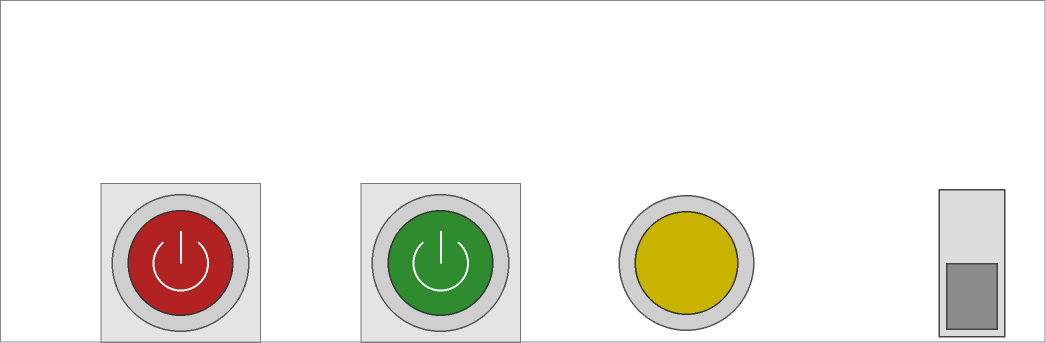
VISUALIZATION Visualization  // 1046x343
    PowerSwitch (83,183 195x160), variable: MAIN.bStopButton, behaviour: TOGGLE, style: Switch-PowerSwitch-Red
    PowerSwitch (343,183 195x160), variable: MAIN.bStartButton, behaviour: TOGGLE, style: Switch-PowerSwitch-Green
    Lamp1 (608,183 157x160), variable: MAIN.bMotor, style: Lamp-Lamp1-Yellow
    DipSwitch (898,183 148x160), variable: MAIN.bLimitSwitch, behaviour: TOGGLE, style: Switch-DipSwitch-Gray
END_VISUALIZATION

(* stored: Version 1.1.0.1
   Visu Visualization: Id {09181a7e-3931-4675-a519-309d1d543899} *)
